// TIA Portal V18 export
FUNCTION_BLOCK "artLimiter"   // FB73, FBD
{ S7_Optimized_Access := 'TRUE' }
VERSION : 0.1
// stored: AutoNumber true, IsIECCheckEnabled false, IsRetainMemResEnabled false, MemoryReserve 100, SetENOAutomatically false, UDAEnableTagReadback false
   VAR_INPUT
      AckEr : Bool;
      UseArtLimitw : Bool;
      artLimfwd : Real;
      artLimRev : Real;
      para_in : "typeMotPara";
   END_VAR
   VAR_OUTPUT
      para_Artlimits : "typeMotPara";
      ER_WS : WString;
      ER : Bool;
   END_VAR
   VAR CONSTANT
      ER_WSlimfwdrev : WString := WSTRING#'art lim rev>fwd';
   END_VAR
BEGIN

REGION Network 1
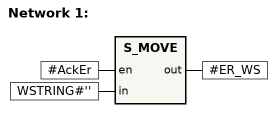
   IF #AckEr THEN #ER_WS := WSTRING#''; END_IF;
END_REGION

REGION Network 2 (SCL)

   #para_Artlimits := #para_in;
   #ER := false;
   IF #artLimfwd < #artLimRev THEN
       #ER_WS := #ER_WSlimfwdrev;
       #ER := true;
   ELSIF #UseArtLimitw THEN
       #para_Artlimits.pos_lim_fwd_USER := MIN(IN1 := #para_in.pos_lim_fwd_USER, IN2 := #artLimfwd);
       #para_Artlimits.pos_lim_rev_USER := MAX(IN1 := #para_in.pos_lim_rev_USER, IN2 := #artLimRev);
   END_IF;
END_REGION
END_FUNCTION_BLOCK
